// TwinCAT 3 PLC project PLC
// ProgramVersion: 3.1.4024.0
// libraries:
//   Tc2_Standard, * (Beckhoff Automation GmbH)
//   Tc2_System, * (Beckhoff Automation GmbH)
//   Tc3_Module, * (Beckhoff Automation GmbH)
// project tree:
//   DUTs/ ST_AxisFault.TcDUT
//   GVLs/ GVL.TcGVL
//   / PlcTask.TcTTO
//   POUs/ FB_Axis.TcPOU, MAIN.TcPOU
// real-time tasks:
//   TASK PlcTask: cycle T#10ms, priority 20, ADS port 350

CONFIGURATION PLC
    RESOURCE PLC ON TwinCAT3
        TASK PlcTask(INTERVAL := T#10ms, PRIORITY := 20);
        PROGRAM MAIN WITH PlcTask : MAIN;
    END_RESOURCE
END_CONFIGURATION

// ---- DUTs/ST_AxisFault.TcDUT
TYPE ST_AxisFault :
STRUCT
	bMcPowerOff		: BOOL;
	bOverCurrent	: BOOL;
	bSTO			: BOOL;
END_STRUCT
END_TYPE

// ---- GVLs/GVL.TcGVL
{attribute 'qualified_only'}
VAR_GLOBAL
	Axes		: ARRAY[0..4] OF FB_Axis;
	AxesFaults	: ARRAY[0..4] OF ST_AxisFault;
END_VAR

// ---- POUs/MAIN.TcPOU
PROGRAM MAIN
VAR
	i		: DINT;
END_VAR

FOR i := 0 TO 4 DO 
	GVL.Axes[i]();
END_FOR

END_PROGRAM

// ---- POUs/FB_Axis.TcPOU
FUNCTION_BLOCK FB_Axis
VAR_INPUT
END_VAR
VAR_OUTPUT
END_VAR
VAR
	bJogFwd			: BOOL;
	bJogRev			: BOOL;
	bFaulted		: BOOL;
	fPosition		: LREAL;
	fVelocity		: LREAL;
END_VAR

IF bJogFwd THEN
	fVelocity := 10.0;
	fPosition := fPosition + 0.1;
ELSE
	fVelocity := 0;
END_IF

IF bJogRev THEN
	fVelocity := -10.0;
	fPosition := fPosition - 0.1;
ELSE
	fVelocity := 0;
END_IF

END_FUNCTION_BLOCK
